TYPE T_CodeBRAND : STRING[9];
END_TYPE

(* stored: Version 1.1.0.1
   DUT T_CodeBRAND: Id {553fc2ea-4099-4c57-8fc2-fa2f171dc2b9} *)
